// TwinCAT 3 PLC project TimesTest
// ProgramVersion: 3.1.4024.0
// libraries:
//   Tc2_Standard, * (Beckhoff Automation GmbH)
//   Tc3_Module, * (Beckhoff Automation GmbH)
//   TcUnit, * (www.tcunit.org)
//   Times, * (TomasRompotl)
// project tree:
//   Clocks/ PeriodicTriggerTest.TcPOU
//   Convert/ ConvertFunctionsTest.TcPOU
//   / PlcTask.TcTTO, PRG_Test.TcPOU (not stored)
// (motion and I/O tree: see PLC project typestest)
// real-time tasks:
//   TASK TypesTestTask: cycle T#1ms, priority 20, ADS port 350
//   TASK StringsTestTask: cycle T#1ms, priority 21, ADS port 351
//   TASK DataTestTask: cycle T#1ms, priority 22, ADS port 352
//   TASK MathTestTask: cycle T#1ms, priority 23, ADS port 353
//   TASK TimesTestTask: cycle T#1ms, priority 24, ADS port 354

CONFIGURATION TimesTest
    RESOURCE PLC ON TwinCAT3
        TASK PlcTask(INTERVAL := T#1ms, PRIORITY := 24);
        PROGRAM PRG_Test WITH PlcTask : PRG_Test;
    END_RESOURCE
END_CONFIGURATION

// ---- Clocks/PeriodicTriggerTest.TcPOU
FUNCTION_BLOCK PeriodicTriggerTest EXTENDS FB_TestSuite
VAR
END_VAR

KeepDisabled();
TriggerWith10msPeriod();
TriggerWith10msPeriodAndPulseAtStart();

METHOD KeepDisabled
VAR
END_VAR
VAR_INST
	pt : PeriodicTrigger := (Enable := FALSE, Period := T#200MS);
	timer : TON := (IN := TRUE, PT := T#1S);
	wasOn : BOOL;
END_VAR
TcUnit.TEST('Keep disabled');

pt.Cyclic();
wasOn S= pt.Trigger;

timer();
IF (timer.Q) THEN
	timer.IN := FALSE;
	
	AssertEquals_BOOL(
		Expected := FALSE,
		Actual := wasOn,
		Message := 'Periodic trigger triggered when not enabled.'
	);
	
	TEST_FINISHED();
END_IF
END_METHOD

// Test has to be run with 1 ms cycle time
METHOD TriggerWith10msPeriod
VAR
END_VAR
VAR_INST
	pt : PeriodicTrigger := (Enable := TRUE, Period := T#10MS);
	expected : ARRAY[0..40] OF BOOL;
	actual : ARRAY[0..40] OF BOOL;
	cycle : INT := 0;
	init : BOOL := TRUE;
END_VAR
VAR CONSTANT
	EndCycle : INT := 40;
END_VAR
TcUnit.TEST('Trigger with 10 ms period');

IF (init) THEN
	init := FALSE;
	expected[10] := TRUE;
	expected[20] := TRUE;
	expected[30] := TRUE;
END_IF

pt.Cyclic();

IF (cycle < EndCycle) THEN 
	actual[cycle] := pt.Trigger;
	cycle := cycle + 1;

	IF (cycle = EndCycle) THEN
		
		AssertArrayEquals_BOOL(
			Expecteds := expected,
			Actuals := actual,
			Message := 'Periodic trigger should trigger at start of each period after the starting one.'
		);
		
		TEST_FINISHED();
	END_IF
END_IF
END_METHOD

// Test has to be run with 1 ms cycle time
METHOD TriggerWith10msPeriodAndPulseAtStart
VAR
END_VAR
VAR_INST
	pt : PeriodicTrigger := (Enable := TRUE, Period := T#10MS, PulseAtStart := TRUE);
	expected : ARRAY[0..40] OF BOOL;
	actual : ARRAY[0..40] OF BOOL;
	cycle : INT := 0;
	init : BOOL := TRUE;
END_VAR
VAR CONSTANT
	EndCycle : INT := 40;
END_VAR
TcUnit.TEST('Trigger with 10 ms period and pulse at start');

IF (init) THEN
	init := FALSE;
	expected[0] := TRUE;
	expected[10] := TRUE;
	expected[20] := TRUE;
	expected[30] := TRUE;
END_IF

pt.Cyclic();

IF (cycle < EndCycle) THEN 
	actual[cycle] := pt.Trigger;
	cycle := cycle + 1;

	IF (cycle = EndCycle) THEN
		
		AssertArrayEquals_BOOL(
			Expecteds := expected,
			Actuals := actual,
			Message := 'Periodic trigger should trigger at start of each period including the starting one.'
		);
		
		TEST_FINISHED();
	END_IF
END_IF
END_METHOD

END_FUNCTION_BLOCK

// ---- Convert/ConvertFunctionsTest.TcPOU
FUNCTION_BLOCK ConvertFunctionsTest EXTENDS FB_TestSuite
VAR
END_VAR

SecondsToTimeFunction();
TimeToSecondsFunction();

METHOD SecondsToTimeFunction
VAR_INPUT
END_VAR
TcUnit.TEST('SecondsToTime function');

AssertEquals_TIME(
	Expected := T#5S,
	Actual := SecondsToTime(5),
	Message := 'Converted time is not correct'
);

TEST_FINISHED();
END_METHOD

METHOD TimeToSecondsFunction
VAR_INPUT
END_VAR
TcUnit.TEST('TimeToSeconds function');

AssertEquals_LREAL(
	Expected := 5,
	Actual := TimeToSeconds(T#5S),
	Delta := 0,
	Message := 'Converted seconds are not correct'
);

TEST_FINISHED();
END_METHOD

END_FUNCTION_BLOCK
